{attribute 'qualified_only'}
{attribute 'strict'}
TYPE MS :
(
	Init_delay,
	Initialization,
	Start,
	Restart,
	NewTable_DB,
	Write_DB,
	FRANKA_Pick_and_place_PCB,
	FRANKA_Measure,
	LED_confirmation,
	FRANKA_Place_PCB,
	DB_Write,
	Measurement_counter,
	Reset,
	FRANKA_ERROR,
	measurebackup,
	Wait
	
);
END_TYPE

(* stored: Version 1.1.0.1, ProductVersion 3.1.4024.3
   EnumerationTextList MS: Id {dc9d61d2-37ff-4b85-b3a3-fca7f4f336fb} *)
